{attribute 'qualified_only'}
{attribute 'strict'}
TYPE E_MbPoll :
(
	Fast := 0,
	Slow,
	Off
);
END_TYPE

(* stored: Version 1.1.0.1
   DUT E_MbPoll: Id {ceafec89-ebe5-4525-85ee-e0c3ee45996a} *)
